(* Schneider Machine Expert - Basic project Raihan Nagib_Boiler Ladder Diagram, file version 2.7.0.0 *)
(* ProjectInformations: Name=New project *)

HARDWARE
  Cpu 0: TM221CE24R
  ModuleExtensionObject 0: TM3AI8/G
  EthernetConfiguration: NetworkName=M221, IpAllocationMode=FixedAddress, IpAddress=0.0.0.0, SubnetMask=0.0.0.0
  SerialLineConfiguration: Baud=Baud19200, Parity=ParityEven, DataBits=DataBits8, StopBits=StopBits1, PhysicalMedium=PhysicalMediumRs485, TransmissionMode=TransmissionModeModbusRtu, SlaveId=1, Addressing=SlaveAddressing
  MastTask: UsePeriodScanMode=false, PeriodScan=100
  FastTask: Period=255
  CpuBehavior: StartingMode=StartAsPreviousState, AutoSaveRamOnEeprom=true, WatchdogPeriod=250

SYMBOLS  (address, symbol, comment, settings)
  %M0       START_BUTTON
  %M1       STOP_BUTTON
  %M2       MOTOR_STATUS
  %M3       LEVEL_STATUS
  %M4       LIMIT_SWITCH
  %M5       PP01_PRESSURE_PUMP
  %M6       PP02_PRESSURE_PUMP
  %M7       SV01_SOLENOID_VALVE
  %M8       SV02_SOLENOID_VALVE
  %M9       HT01_HEATER
  %M10      HT02_HEATER
  %M11      WP01_WATER_PUMP
  %M12      WP02_WATER_PUMP
  %MW0      PT01_PRESSURE_TRANSMITTER
  %MW1      PT02_PRESSURE_TRANSMITTER
  %MW2      TT01_TEMPERATURE_TRANSMITTER
  %MW3      TT02_TEMPERATURE_TRANSMITTER
  %MW4      FT01_FLOW_TRANSMITTER
  %MW5      FT02_FLOW_TRANSMITTER
  %MW6      WLT01_WATER_LEVEL_TRANSMITTER
  %MW7      WLT02_WATER_LEVEL_TRANSMITTER
  %MW8      LT01_PV_LEVEL_TRANSMITTER
  %MW9      LT01_SP_LEVEL_TRANSMITTER
  %TM0        [Preset=3, Base=OneSecond]

POU New POU
  (* SectionNumber=1 *)

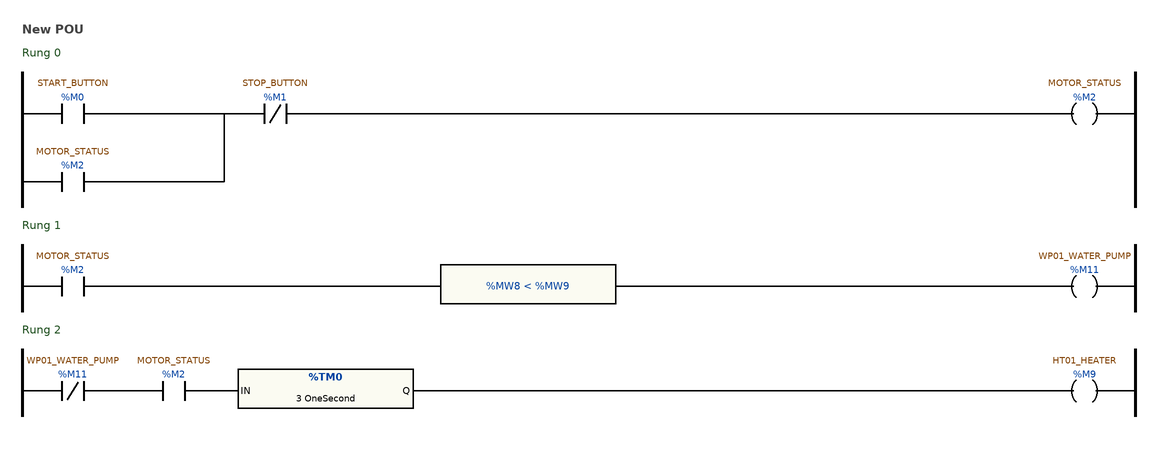

// Rung 0
  LD %M0                  (* START_BUTTON *)
  OR %M2                  (* MOTOR_STATUS *)
  ANDN %M1                (* STOP_BUTTON *)
  ST %M2                  (* MOTOR_STATUS *)
  // as ST:
  //   MOTOR_STATUS := (START_BUTTON OR MOTOR_STATUS) AND NOT STOP_BUTTON;

// Rung 1
  LD %M2                  (* MOTOR_STATUS *)
  AND [ %MW8 < %MW9 ]     (* LT01_PV_LEVEL_TRANSMITTER, LT01_SP_LEVEL_TRANSMITTER *)
  ST %M11                 (* WP01_WATER_PUMP *)
  // as ST:
  //   WP01_WATER_PUMP := MOTOR_STATUS AND LT01_PV_LEVEL_TRANSMITTER < LT01_SP_LEVEL_TRANSMITTER;

// Rung 2
  BLK %TM0
  LDN %M11                (* WP01_WATER_PUMP *)
  AND %M2                 (* MOTOR_STATUS *)
  IN
  OUT_BLK
  LD Q
  ST %M9                  (* HT01_HEATER *)
  END_BLK
  // as ST:
  //   %TM0(IN := NOT WP01_WATER_PUMP AND MOTOR_STATUS);
  //   HT01_HEATER := %TM0.Q;
